FUNCTION IntegerToBoolArray : BOOL
VAR_IN_OUT
	arr : ARRAY[*] OF BOOL;
END_VAR
VAR_INPUT
	num : ULINT;
END_VAR
VAR_OUTPUT
	maxIterations : DINT;
END_VAR
VAR
	i : DINT;
	j : LINT;
END_VAR

maxIterations := MIN(
	(UPPER_BOUND(arr,1) - LOWER_BOUND(arr,1) + 1),
	SIZEOF(num) * 8);

FOR i:=LOWER_BOUND(arr, 1) TO UPPER_BOUND(arr, 1) BY 1 DO
	IF j < maxIterations THEN
		arr[i] := IntegerBitAccess(num, j);
		j := j + 1;
	END_IF
END_FOR

END_FUNCTION

(* stored: Version 1.1.0.1, ProductVersion 3.1.4024.11
   POU IntegerToBoolArray: Id {0b5a855f-d726-46ed-b13f-e23c9348216a}, SpecialFunc None *)
